FUNCTION_BLOCK E_INIT_CHK_D (* Sends INIT event the first time a REQ event arrives and a NOINIT event for every subsequent REQ event. *)
  (* Standard: 61499-2 *)
  (* Version 1.0, 2017-06-17, Marc Jakobi, HTW Berlin *)
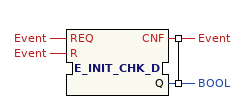
  EVENT_INPUT
    REQ; (* Normal Execution Request *)
    R; (* Reset *)
  END_EVENT
  EVENT_OUTPUT
    CNF WITH Q; (* Confirmation Event *)
  END_EVENT
  VAR_OUTPUT
    Q : BOOL; (* true if first time REQ arrived, false otherwise *)
  END_VAR
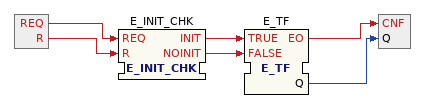
  FBS
    E_INIT_CHK : E_INIT_CHK;
    E_TF : E_TF;
  END_FBS
  EVENT_CONNECTIONS
    REQ TO E_INIT_CHK.REQ;
    R TO E_INIT_CHK.R;
    E_TF.EO TO CNF;
    E_INIT_CHK.INIT TO E_TF.TRUE;
    E_INIT_CHK.NOINIT TO E_TF.FALSE;
  END_CONNECTIONS
  DATA_CONNECTIONS
    E_TF.Q TO Q;
  END_CONNECTIONS
END_FUNCTION_BLOCK
